FUNCTION invMat7 : bool
VAR_IN_OUT CONSTANT
	mat :Mat7d;
END_VAR

VAR_IN_OUT
	invMat :Mat7d;
END_VAR
VAR
	dim : INT :=7;
	i,j,k,h:INT;
	m,n :INT;
	cofactorMat : Mat6d;
	adjointMat :Mat7d;
	matDet :LREAL;
END_VAR

matDet :=Det7(mat);
IF matDet=0 THEN
	invMat7:=FALSE;
	RETURN;
END_IF

FOR i :=1 TO dim DO
	FOR j:=1 TO dim DO
		// get cofactor mat
		m:=1;
		n:=1;
		FOR k:=1 TO dim DO
			FOR h:=1 TO dim DO
				IF k<>i AND h <> j THEN
					cofactorMat[m,n]:=mat[k,h];
					n:=n+1;
					IF n>=dim THEN
						m:=m+1;
						n:=1;
					END_IF
				END_IF
			END_FOR
		END_FOR
		
		adjointMat[i,j]:=EXPT(-1,i+j)*Det6(cofactorMat);
	END_FOR
END_FOR

FOR i :=1 TO dim DO
	FOR j:=1 TO dim DO
		invMat[i,j]:=adjointMat[j,i]/matDet;
	END_FOR
END_FOR
invMat7:=true;

END_FUNCTION

(* stored: Version 1.1.0.1, ProductVersion 3.1.4024.12
   POU invMat7: Id {e60c154b-d5c5-461b-abce-ac90f00b4245}, SpecialFunc None *)
